KUKA KRL program: DROOP_PALL.src, DROOP_PALL.dat

--- DROOP_PALL.src ---
&ACCESS RVO2
&REL 52
&PARAM EDITMASK = *
&PARAM TEMPLATE = C:\KRC\Roboter\Template\vorgabe
&PARAM DISKPATH = KRC:\R1\Program\R_02
DEF DROOP_PALL( )
;FOLD INI;%{PE}
  ;FOLD BASISTECH INI
    GLOBAL INTERRUPT DECL 3 WHEN $STOPMESS==TRUE DO IR_STOPM ( )
    INTERRUPT ON 3
    BAS (#INITMOV,0 )
  ;ENDFOLD (BASISTECH INI)
  ;FOLD USER INI
    ;Make your modifications here

  ;ENDFOLD (USER INI)
;ENDFOLD (INI)

INTERRUPT DECL 21 WHEN  i_Paleta_POZ == FALSE DO IR_MOVESTOP()  ;Stop odlozenia palety na stos

;wykomentowany
;FOLD PTP HOME Vel=100 % DEFAULT;%{PE}
;FOLD Parameters ;%{h}
;Params IlfProvider=kukaroboter.basistech.inlineforms.movement.old; Kuka.IsGlobalPoint=False; Kuka.PointName=HOME; Kuka.BlendingEnabled=False; Kuka.MoveDataPtpName=DEFAULT; Kuka.VelocityPtp=100; Kuka.CurrentCDSetIndex=0; Kuka.MovementParameterFieldEnabled=True; IlfCommand=PTP
;ENDFOLD
$BWDSTART = FALSE
PDAT_ACT = PDEFAULT
FDAT_ACT = FHOME
BAS(#PTP_PARAMS, 100.0)
SET_CD_PARAMS (0)
;PTP XHOME
;ENDFOLD


;wykomentowany
XTO_PAL_DROOP_05={X -45.0, Y 250.0, Z 2100.0, A -90, B 0.0, C 180}
;FOLD PTP TO_PAL_DROOP_05 CONT Vel=100 % PDATH Tool[2]:TCP_PALETA Base[5]:ODLOZENIE_PALETY;%{PE}
;FOLD Parameters ;%{h}
;Params IlfProvider=kukaroboter.basistech.inlineforms.movement.old; Kuka.IsGlobalPoint=False; Kuka.PointName=TO_PAL_DROOP_05; Kuka.BlendingEnabled=True; Kuka.MoveDataPtpName=PDATH; Kuka.VelocityPtp=100; Kuka.CurrentCDSetIndex=0; Kuka.MovementParameterFieldEnabled=True; IlfCommand=PTP
;ENDFOLD
$BWDSTART = FALSE
PDAT_ACT = PPDATH
FDAT_ACT = FTO_PAL_DROOP_05
BAS(#PTP_PARAMS, 100.0)
SET_CD_PARAMS (0)
; PTP XTO_PAL_DROOP_05 C_Dis
;ENDFOLD

WAIT FOR  i_Paleta_POZ

XPRE_PAL_DROOP={X 0.0,Y 0.0,Z 2100.0,A -90.0,B 0.0,C 180.0,S 2, T 11}
;FOLD PTP PRE_PAL_DROOP CONT Vel=100 % PDATH Tool[2]:TCP_PALETA Base[5]:ODLOZENIE_PALETY;%{PE}
;FOLD Parameters ;%{h}
;Params IlfProvider=kukaroboter.basistech.inlineforms.movement.old; Kuka.IsGlobalPoint=False; Kuka.PointName=PRE_PAL_DROOP; Kuka.BlendingEnabled=True; Kuka.MoveDataPtpName=PDATH; Kuka.VelocityPtp=100; Kuka.CurrentCDSetIndex=0; Kuka.MovementParameterFieldEnabled=True; IlfCommand=PTP
;ENDFOLD
$BWDSTART = FALSE
PDAT_ACT = PPDATH
FDAT_ACT = FPRE_PAL_DROOP
BAS(#PTP_PARAMS, 100.0)
SET_CD_PARAMS (0)
PTP XPRE_PAL_DROOP C_Dis
;ENDFOLD

;Odlozenie palety
XPAL_DROOP={X 0.0,Y 0.0,Z 50.0,A -90.0,B 0.0,C 180.0,S 2, T 11}
Fpozy2 = FPAL_DROOP
Xpozy2 = XPAL_DROOP

INTERRUPT ON 21
Ruch_W_Dol(0.5) ; zjazd w dol
INTERRUPT OFF 21
$ADVANCE=3

;FOLD Gripper SET [3]widly_paleta State=[1]OPEN Wait 0.2[s] Check with Strategy 1 ;%{PE}
;FOLD Parameters Parameters ;%{h}
;Params IlfProvider=GripperTech.GripperSet;setgripper=3;setstate=1;setcont=nocont;waittime=0.2;errorstrategy=1
;ENDFOLD
GRPg_SetStateAndCheck(3, 1, 0.2, 1)
;ENDFOLD

XPAL_POST_DROOP=$POS_ACT
XPAL_POST_DROOP.Z=XPAL_POST_DROOP.Z+100
;FOLD LIN PAL_POST_DROOP Vel=1 m/s LDATM Tool[2]:TCP_PALETA Base[5]:ODLOZENIE_PALETY ;%{PE}
;FOLD Parameters ;%{h}
;Params IlfProvider=kukaroboter.basistech.inlineforms.movement.old; Kuka.IsGlobalPoint=False; Kuka.PointName=PAL_POST_DROOP; Kuka.BlendingEnabled=False; Kuka.MoveDataName=LDATM; Kuka.VelocityPath=1; Kuka.CurrentCDSetIndex=0; Kuka.MovementParameterFieldEnabled=True; IlfCommand=LIN
;ENDFOLD
$BWDSTART = FALSE
LDAT_ACT = LLDATM
FDAT_ACT = FPAL_POST_DROOP
BAS(#CP_PARAMS, 1.0)
SET_CD_PARAMS (0)
LIN XPAL_POST_DROOP
;ENDFOLD

;FOLD PTP PRE_PAL_DROOP CONT Vel=100 % PDATH Tool[2]:TCP_PALETA Base[5]:ODLOZENIE_PALETY;%{PE}
;FOLD Parameters ;%{h}
;Params IlfProvider=kukaroboter.basistech.inlineforms.movement.old; Kuka.IsGlobalPoint=False; Kuka.PointName=PRE_PAL_DROOP; Kuka.BlendingEnabled=True; Kuka.MoveDataPtpName=PDATH; Kuka.VelocityPtp=100; Kuka.CurrentCDSetIndex=0; Kuka.MovementParameterFieldEnabled=True; IlfCommand=PTP
;ENDFOLD
$BWDSTART = FALSE
PDAT_ACT = PPDATH
FDAT_ACT = FPRE_PAL_DROOP
BAS(#PTP_PARAMS, 100.0)
SET_CD_PARAMS (0)
PTP XPRE_PAL_DROOP C_Dis
;ENDFOLD


;FOLD PTP HOME Vel=100 % DEFAULT;%{PE}
;FOLD Parameters ;%{h}
;Params IlfProvider=kukaroboter.basistech.inlineforms.movement.old; Kuka.IsGlobalPoint=False; Kuka.PointName=HOME; Kuka.BlendingEnabled=False; Kuka.MoveDataPtpName=DEFAULT; Kuka.VelocityPtp=100; Kuka.CurrentCDSetIndex=0; Kuka.MovementParameterFieldEnabled=True; IlfCommand=PTP
;ENDFOLD
$BWDSTART = FALSE
PDAT_ACT = PDEFAULT
FDAT_ACT = FHOME
BAS(#PTP_PARAMS, 100.0)
SET_CD_PARAMS (0)
PTP XHOME
;ENDFOLD

END

DEF IR_MOVESTOP()
  INTERRUPT OFF 21 ;BRAKE MOVEMENT DIRECTION
    BRAKE
    RESUME
;  HALT ; Dla testu odkomentowac

END

DEF Ruch_W_Dol(SPEED:IN)
DECL REAL SPEED

$BWDSTART = FALSE
LDAT_ACT=LLDAT0
FDAT_ACT=Fpozy2
BAS(#CP_PARAMS,SPEED)
LIN Xpozy2

$ADVANCE = 0
END

--- DROOP_PALL.dat ---
&ACCESS RVO2
&REL 52
&PARAM EDITMASK = *
&PARAM TEMPLATE = C:\KRC\Roboter\Template\vorgabe
&PARAM DISKPATH = KRC:\R1\Program\R_02
DEFDAT  DROOP_PALL
;FOLD EXTERNAL DECLARATIONS;%{PE}%MKUKATPBASIS,%CEXT,%VCOMMON,%P
;FOLD BASISTECH EXT;%{PE}%MKUKATPBASIS,%CEXT,%VEXT,%P
EXT  BAS (BAS_COMMAND  :IN,REAL  :IN )
DECL INT SUCCESS
;ENDFOLD (BASISTECH EXT)
;FOLD USER EXT;%{E}%MKUKATPUSER,%CEXT,%VEXT,%P
;Make your modifications here

;ENDFOLD (USER EXT)
;ENDFOLD (EXTERNAL DECLARATIONS)

;SIGNAL data
SIGNAL i_Paleta_POZ $IN[147] ;Czujnik wykrycia palety

;E6POS data
DECL E6POS Xpozy2
DECL E6POS XPAL_DROOP
DECL E6POS XPRE_PAL_DROOP
DECL E6POS XTO_PAL_DROOP
DECL E6POS XPAL_POST_DROOP
DECL E6POS XTO_PAL_DROOP_05={X -45.0000,Y 250.000,Z 2100.00,A -90.0000,B 0.0,C 180.000}

;FDAT data
DECL FDAT Fpozy2={TOOL_NO 2,BASE_NO 5,IPO_FRAME #BASE,POINT2[] " "}
DECL FDAT FTO_PAL_DROOP={TOOL_NO 2,BASE_NO 5,IPO_FRAME #BASE,POINT2[] " "}
DECL FDAT FPRE_PAL_DROOP={TOOL_NO 2,BASE_NO 5,IPO_FRAME #BASE,POINT2[] " "}
DECL FDAT FPAL_DROOP={TOOL_NO 2,BASE_NO 5,IPO_FRAME #BASE,POINT2[] " "}
DECL FDAT FPAL_POST_DROOP={TOOL_NO 2,BASE_NO 5,IPO_FRAME #BASE,POINT2[] " "}
DECL FDAT FTO_PAL_DROOP_05={TOOL_NO 2,BASE_NO 5,IPO_FRAME #BASE,POINT2[] " "}

;LDAT data
DECL LDAT LLDAT0={VEL 0.200000,ACC 100.000,APO_DIST 100.000,APO_FAC 50.0000,ORI_TYP #VAR}
DECL LDAT LLDATM={VEL 1.00000,ACC 100.000,APO_DIST 100.000,APO_FAC 50.0000,AXIS_VEL 100.000,AXIS_ACC 100.000,ORI_TYP #VAR,CIRC_TYP #BASE,JERK_FAC 50.0000,GEAR_JERK 100.000,EXAX_IGN 0}

;PDAT data
DECL PDAT PPDATH={VEL 100.000,ACC 100.000,APO_DIST 100.000,APO_MODE #CDIS,GEAR_JERK 100.000,EXAX_IGN 0}

;MODULE
DECL MODULEPARAM_T LAST_TP_PARAMS={PARAMS[] "Kuka.VelocityPtp=100; Kuka.BlendingEnabled=False; Kuka.CurrentCDSetIndex=0    "}
ENDDAT
